// TIA Portal V17 export
// export: Created 2025-06-20T12:46:57.9079355Z, ExportSetting WithDefaults, DisplayName Totally Integrated Automation Portal, DisplayVersion V17 Update 8, DisplayName TIA Portal Openness, DisplayVersion V17 Update 8, DisplayName TIA Portal Version Control Interface, DisplayVersion V17, DisplayName SINAMICS Startdrive Advanced, DisplayVersion V17 SP2, DisplayName SINAMICS Startdrive G110M, G120, G120C, G120D, G120P, G115D, DisplayVersion V17 SP2, DisplayName SINAMICS Startdrive G130, G150, S120, S150, SINAMICS MV, S210, DisplayVersion V17 SP2, DisplayName STEP 7 Professional, DisplayVersion V17 Update 8, DisplayName SINUMERIK ONE STEP 7 Toolbox, DisplayVersion V17 Update 12, DisplayName SINUMERIK ONE PLC Basic Program Plus, DisplayVersion V17 Update 12, DisplayName SINUMERIK 840D sl STEP 7 Toolbox, DisplayVersion V17 Update 12, DisplayName STEP 7 Safety, DisplayVersion V17 Update 6, DisplayName WinCC Advanced, DisplayVersion V17 Update 8
DATA_BLOCK "DB16225_RELEASE_HANDLE_LIST_U2_STA2_MEAS"   // DB16225
{ DB_Accessible_From_OPC_UA := 'FALSE' }
// stored: AutoNumber false, DBAccessibleFromOPCUA false, DBAccessibleFromWebserver true, InstanceOfName OPC_UA_NodeReleaseHandleList, OfSystemLibElement OPC_UA_NodeReleaseHandleList, OfSystemLibVersion 1.0
"OPC_UA_NodeReleaseHandleList"
   // VAR_INPUT
   //    REQ : Bool;
   //    ConnectionHdl : DWord;
   //    NodeHdlCount : UInt;
   //    NodeHdls : Variant;
   //    Timeout : Time;
   // END_VAR
   // VAR_OUTPUT
   //    Done : Bool;
   //    Busy : Bool;
   //    Error : Bool;
   //    Status : DWord;
   // END_VAR
   // VAR_IN_OUT
   //    NodeStatusList : Variant;
   // END_VAR
BEGIN
END_DATA_BLOCK
